FUNCTION_BLOCK oneComposite (* Composite FB wrapping other FBs *)
  (* Standard: 61499-2 *)
  (* Version 1.0, 2022-08-01, franz *)
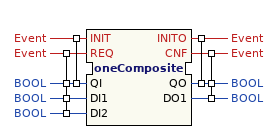
  EVENT_INPUT
    INIT WITH QI; (* Initialization Request *)
    REQ WITH QI, DI1, DI2; (* Normal Execution Request *)
  END_EVENT
  EVENT_OUTPUT
    INITO WITH QO; (* Initialization Confirm *)
    CNF WITH QO, DO1; (* Execution Confirmation *)
  END_EVENT
  VAR_INPUT
    QI : BOOL; (* Input event qualifier *)
    DI1 : BOOL;
    DI2 : BOOL;
  END_VAR
  VAR_OUTPUT
    QO : BOOL; (* Output event qualifier *)
    DO1 : BOOL;
  END_VAR
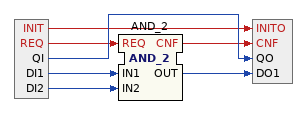
  FBS
    AND_2 : AND_2;
  END_FBS
  EVENT_CONNECTIONS
    REQ TO AND_2.REQ;
    AND_2.CNF TO CNF;
    INIT TO INITO;
  END_CONNECTIONS
  DATA_CONNECTIONS
    DI1 TO AND_2.IN1;
    DI2 TO AND_2.IN2;
    AND_2.OUT TO DO1;
    QI TO QO;
  END_CONNECTIONS
END_FUNCTION_BLOCK
